FUNCTION_BLOCK PUBLIC FB_LTU EXTENDS FB_IndexedPosition

VAR_IN_OUT
	HardwareInputArray : ARRAY [*] OF BOOL;		// For Actuators
END_VAR

VAR
	Configuration 		: ST_LTUConfiguration;
	Status				: ST_LTUStatus;
	
	InitDone 			: BOOL := FALSE;

	LTUHardwareState	: DINT := E_LTUHardwareState.NoCommand;
END_VAR

IF NOT InitDone THEN
	M_Init();
	InitDone:= TRUE;
ELSE
	SUPER^();
	M_Cyclic();
	M_StateMachine();
END_IF

METHOD PRIVATE M_Cyclic : BOOL
VAR_INPUT
END_VAR
Controls.isDefined := TRUE; // I exist

Configuration.ForwardOutputArrayPosition 	:= Configuration.ForwardHardwareOutput - 32768;
Configuration.ReverseOutputArrayPosition 	:= Configuration.ReverseHardwareOutput - 32768;
Configuration.LeftOutputArrayPosition 		:= Configuration.LeftHardwareOutput - 32768;
Configuration.RightOutputArrayPosition 		:= Configuration.RightHardwareOutput - 32768;

HardwareInputArray[Configuration.ForwardOutputArrayPosition] 	:= SEL( LTUHardwareState = E_LTUHardwareState.RunForward, FALSE, TRUE);
HardwareInputArray[Configuration.ReverseOutputArrayPosition] 	:= SEL( LTUHardwareState = E_LTUHardwareState.RunReverse, FALSE, TRUE);
HardwareInputArray[Configuration.LeftOutputArrayPosition] 		:= SEL( LTUHardwareState = E_LTUHardwareState.RunLeft, FALSE, TRUE);
HardwareInputArray[Configuration.RightOutputArrayPosition] 		:= SEL( LTUHardwareState = E_LTUHardwareState.RunRight, FALSE, TRUE);
END_METHOD

METHOD PRIVATE M_Init : BOOL
VAR_INPUT
END_VAR
END_METHOD

METHOD PUBLIC M_Reset : BOOL
VAR_INPUT
END_VAR
LTUHardwareState := E_LTUHardwareState.NoCommand;

SUPER^.P_Controls.Front.Request := E_IndexedPositionSimplifiedRequest.NoRequest;
SUPER^.P_Controls.Rear.Request := E_IndexedPositionSimplifiedRequest.NoRequest;
SUPER^.P_Controls.Left.Request := E_IndexedPositionSimplifiedRequest.NoRequest;
SUPER^.P_Controls.Right.Request := E_IndexedPositionSimplifiedRequest.NoRequest;

SUPER^.P_Controls.Request := E_IndexedPositionTransitionRequest.NoRequest;
SUPER^.P_Controls.State := E_IndexedPositionStates.Starved;
END_METHOD

METHOD PRIVATE M_StateMachine : BOOL
VAR_INPUT
END_VAR
(*IF Configuration.BypassLTU THEN
	State := E_LTUStates.Bypass;
ELSE
	State := E_LTUStates.Idle;
END_IF*)

CASE SUPER^.Controls.State OF
	E_IndexedPositionStates.Starved, 
	E_IndexedPositionStates.Idle, 
	E_IndexedPositionStates.Blocked, 
	E_IndexedPositionStates.Fault:
		LTUHardwareState := E_LTUHardwareState.NoCommand;
			
	E_IndexedPositionStates.ReceivingFromRight, 
	E_IndexedPositionStates.SendingToLeft:
		LTUHardwareState := E_LTUHardwareState.RunLeft;

	E_IndexedPositionStates.ReceivingFromLeft, 
	E_IndexedPositionStates.SendingToRight:
		LTUHardwareState := E_LTUHardwareState.RunRight;

	E_IndexedPositionStates.ReceivingFromRear, 
	E_IndexedPositionStates.SendingToFront:
		LTUHardwareState := E_LTUHardwareState.RunForward;
		
	E_IndexedPositionStates.ReceivingFromFront, 
	E_IndexedPositionStates.SendingToRear:
		LTUHardwareState := E_LTUHardwareState.RunReverse;
		
	E_IndexedPositionStates.Bypass:
		LTUHardwareState := E_LTUHardwareState.RunForward;
		
END_CASE
END_METHOD

PROPERTY PUBLIC P_Configuration : REFERENCE TO ST_LTUConfiguration
GET
P_Configuration REF= Configuration;
END_GET
END_PROPERTY

PROPERTY PUBLIC P_Status : REFERENCE TO ST_LTUStatus
GET
P_Status REF= Status;
END_GET
END_PROPERTY

END_FUNCTION_BLOCK

(* stored: Version 1.1.0.1, ProductVersion 3.1.4024.12
   POU FB_LTU: Id {9a3a695d-874f-4a99-a04d-54c171fe4ae2}, SpecialFunc None
   Method M_Cyclic: Id {2c03fa0c-75a0-4d97-94fc-1f4e2d386c87}
   Method M_Init: Id {89a5733f-5226-45aa-aad7-e130af7257fa}
   Method M_Reset: Id {cf69b0fe-4f1e-40da-87ff-22d8542cf7e7}
   Method M_StateMachine: Id {401b7a95-1b5d-4eb7-8b1c-33ec096717ce}
   Property P_Configuration: Id {0f8ff860-f9b3-4c36-a003-5520c8fde47e}
   Get Get: Id {60d5b67b-3c9d-49a5-8918-917adf8a6aae}
   Property P_Status: Id {8e24c6f7-a6a0-4bc6-a85a-a81f7d3f5058}
   Get Get: Id {f8bc7630-fd81-44b1-ae66-983ebbb9446b} *)
